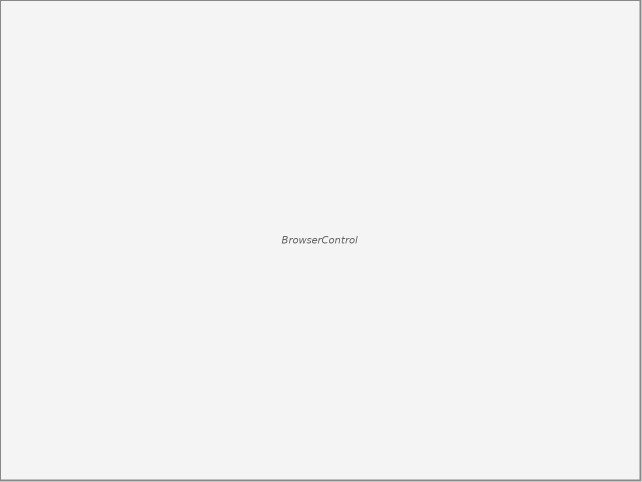
VISUALIZATION vBrowser  // 642x482
    BrowserControl (0,0 640x480)
        p3734058945: 'https://yandex.ru/internet/'
        p2179181546: MAIN.bBrowserStart
END_VISUALIZATION

(* stored: Version 1.1.0.1, ProductVersion 3.1.4024.2
   Visu vBrowser: Id {402b63e7-a696-4504-9f7a-648afcdeb381} *)
